Fanuc KAREL source: kf00097.KL

-- PROVISIONAL review KL for V770-1; original PC SHA256 83a4cbbc1f5960138fe53c78cf5eb845b0c0c2de99f6cf14a1f67f4654d5874e
-- Incomplete behavior may be omitted. Consult companion uncertainty JSON. Do not deploy.
PROGRAM KF00097
%NOLOCKGROUP
BEGIN
  -- UNRESOLVED_PC offsets 5-16; opcodes 2E,23
  -- UNRESOLVED_PC offsets 21-32; opcodes 2E,23
  -- UNRESOLVED_PC offsets 37-55; opcodes 27,27,9D,22,22,31
  -- UNRESOLVED_PC offsets 60-64; opcodes 7F
END KF00097
